Omron CX-Programmer project NewProject (CX-Programmer 9.61)

# PLC NewPLC1: CP1E N30

## Global symbols (name address type ; comment)
0.00 BOOL  ; ON
0.01 BOOL  ; OFF
100.00 BOOL  ; Lampu 1

## Program NewProgram1 (cyclic task 0)

### Section Section1

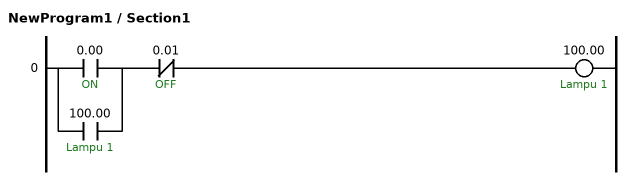
; rung 0
LD 0.00  ; ON
OR 100.00  ; Lampu 1
ANDNOT 0.01  ; OFF
OUT 100.00  ; Lampu 1
; rung 1
END(001)

### Section END
; rung 0
END(001)